PROGRAM MAIN
VAR
	//EM Pallet Transport
	sim_MOVITRAC_B : SIM_MOVITRAC_B;
	sim_MOVITRAC_B2 : SIM_MOVITRAC_B2;
	simCentering : SIM_ValveWithDoubleFB;	

	//EM Docking Interface
	simDockingClampUpper : SIM_ValveWithDoubleFB;
	simDockingClampLower : SIM_ValveWithDoubleFB;
	simUnlockPinUpper : SIM_ValveWithFB;
	simUnlockPinLower : SIM_ValveWithFB;
	simDoorOpener : SIM_ValveWithFB;
	simDoorShutter : SIM_ValveWithFB;
	simDoorOpenerAlmostClosed AT %Q* : BOOL;
	tonDoorOpenerAlmosClosed : TON;
	
	simLiftActPosition AT %I* : LREAL;
	simLiftHomed AT %Q* : BOOL;
	simTransportUnitActPos AT %I* : LREAL;
	simTransportUnitHomed AT %Q* : BOOL;
	
	bInitDone : BOOL;
	simSafetyOK AT %Q* : BOOL;
	simPowerOK AT %Q* : BOOL;
	simAirPressureOK AT %Q* : BOOL;
	
	{attribute 'TcLinkTo' := 'TIPC^CleanroomConnect^CleanroomConnect Instance^PlcTask Outputs^GVL_Modules.g_emPalletConveyor.s_cmPalletConveyor.Q_bCmdReset'}
	I_bCmdReset AT %I* : BOOL;
	{attribute 'TcLinkTo' := 'TIPC^CleanroomConnect^CleanroomConnect Instance^PlcTask Outputs^GVL_Modules.g_emPalletConveyor.s_cmPalletConveyor.Q_bCmdEnable'}
	I_bCmdEnable AT %I* : BOOL;
	{attribute 'TcLinkTo' := 'TIPC^CleanroomConnect^CleanroomConnect Instance^PlcTask Outputs^GVL_Modules.g_emPalletConveyor.s_cmPalletConveyor.Q_bCmdStartCW'}
	I_bCmdStartCW AT %I* : BOOL;
	{attribute 'TcLinkTo' := 'TIPC^CleanroomConnect^CleanroomConnect Instance^PlcTask Outputs^GVL_Modules.g_emPalletConveyor.s_cmPalletConveyor.Q_bCmdStartCCW'}
	I_bCmdStartCCW AT %I* : BOOL;
	{attribute 'TcLinkTo' := 'TIPC^CleanroomConnect^CleanroomConnect Instance^PlcTask Inputs^GVL_Modules.g_emPalletConveyor.s_cmPalletConveyor.I_bStaReadyForOperation'}
	Q_bStaReadyForOperation AT %Q* : BOOL;
	{attribute 'TcLinkTo' := 'TIPC^CleanroomConnect^CleanroomConnect Instance^PlcTask Inputs^GVL_Modules.g_emPalletConveyor.s_cmPalletConveyor.I_bStaMotorIsRunning'}
	Q_bStaMotorIsRunning AT %Q* : BOOL;
	
END_VAR


IF NOT(bInitDone) THEN
	simSafetyOK := TRUE;
	simPowerOK := TRUE;
	simAirPressureOK := TRUE;
	
	simDoorShutter.mForceOff();
	simDoorOpener.mForceOff();
	
	bInitDone := TRUE;
END_IF

//EM Pallet Conveyor
sim_MOVITRAC_B();

sim_MOVITRAC_B2(
	i_ref_I_bCmdReset := I_bCmdReset, 
	i_ref_I_bCmdEnable := I_bCmdEnable, 
	i_ref_I_bCmdStartCW := I_bCmdStartCW, 
	i_ref_I_bCmdStartCCW := I_bCmdStartCCW, 
	i_ref_Q_bStaReadyForOperation := Q_bStaReadyForOperation, 
	i_ref_Q_bStaMotorIsRunning := Q_bStaMotorIsRunning);

simCentering();

//EM Docking Interface
simDockingClampUpper();
simDockingClampLower();
simUnlockPinUpper();
simUnlockPinLower();
simDoorOpener();
simDoorShutter();

tonDoorOpenerAlmosClosed(IN := (simDoorOpener.q_bCmdValveOff OR simDoorOpener.q_bStaValveOff), PT := T#1S);
simDoorOpenerAlmostClosed := tonDoorOpenerAlmosClosed.Q; 

//IF (simLiftActPosition > 9999999000 AND simLiftActPosition < 10000000000 THEN
//simLiftHomed := TRUE;

//simLiftHomed := FALSE;

END_PROGRAM

(* stored: Version 1.1.0.1, ProductVersion 3.1.4024.12
   POU MAIN: Id {81b5c3b0-b471-4cd8-addb-1925034be3d2}, SpecialFunc None *)
